{attribute 'qualified_only'}
{attribute 'strict'}
{attribute 'to_string'}
TYPE E_LIST_CHECK :
(
	NULL,
  REFERENCE_CTRL_INVALID := 9000,
  REFERENCE_STATE_INVALID,
  REFERENCE_DATA_INPUT_INVALID,
  REFERENCE_DATA_OUTPUT_INVALID,

  CHECK_DONE              := 10000
);
END_TYPE

(* stored: Version 1.1.0.1, ProductVersion 3.1.4026.18
   DUT E_LIST_CHECK: Id {f17c9ade-1d49-4056-8427-3ce44cea9ddf} *)
